FUNCTION_BLOCK InitState IMPLEMENTS I_SD_ValveState
VAR_INPUT
END_VAR
VAR_OUTPUT
END_VAR
VAR
    _ptSdValve : POINTER TO SD_Valve;
    _transition : I_Transitive;
    delayTimer : Tc2_Standard.TON;
    start : BOOL;
END_VAR

delayTimer(IN:=start,PT:=T#10S);
IF NOT start THEN
    start := TRUE;
END_IF
IF delayTimer.q THEN
    start := FALSE;
//    _ptSdValve^.GoToAutoState();
    IF _transition<>0 THEN
        _transition.Transit();
	END_IF
END_IF

METHOD Close : BOOL
Close := false;
END_METHOD

METHOD FB_init : BOOL
VAR_INPUT
	bInitRetains : BOOL; // if TRUE, the retain variables are initialized (warm start / cold start)
	bInCopyCode : BOOL;  // if TRUE, the instance afterwards gets moved into the copy code (online change)
    ptSdValve : POINTER TO SD_Valve;
END_VAR
_ptSdValve := ptSdValve;
END_METHOD

METHOD Open : BOOL
Open := False;
END_METHOD

METHOD RUN
THIS^();
END_METHOD

METHOD SetTransition
VAR_INPUT
	transition	: I_Transitive;
END_VAR
_transition := transition;
END_METHOD

PROPERTY StateName : STRING
GET
StateName := 'Init';
END_GET
END_PROPERTY

END_FUNCTION_BLOCK

(* stored: Version 1.1.0.1, ProductVersion 3.1.4024.12
   POU InitState: Id {c6492e7b-2779-484f-91cc-b35751e8ded7}, SpecialFunc None
   Method Close: Id {5e87cd17-9222-4cf5-9066-4ffa84d6ae0b}
   Method FB_init: Id {ebfe7b03-d6f2-4ca9-a28f-4604097172bd}
   Method Open: Id {71edc793-e772-4664-8a7d-02014c800cb4}
   Method RUN: Id {964efa80-522f-4e8d-bd85-9cecd5924c27}
   Method SetTransition: Id {82a09f8e-925f-4ba2-a84e-cfae191e2315}
   Property StateName: Id {db9bba26-be28-4c34-bf48-770d0b2ec75a}
   Get Get: Id {e9684588-bec9-4d32-bcce-84cf4b1356d6} *)
